// Mitsubishi GX Works2 project: 240909_공급가공   PLC: Q03UDV

PROGRAM MAIN
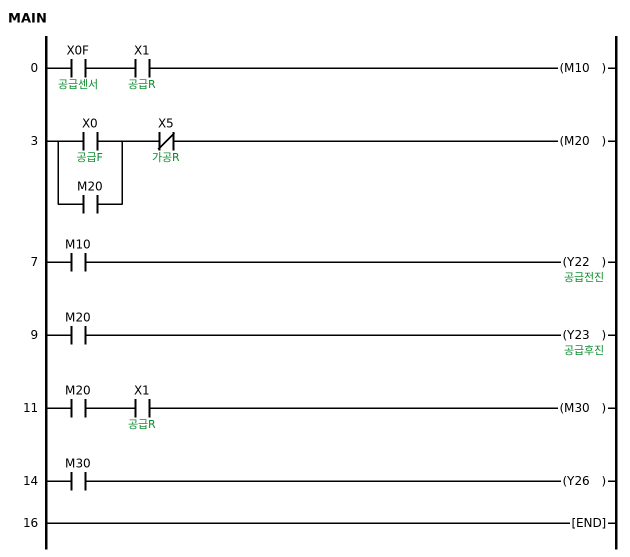
0     LD      X0F  ; 공급센서
      AND     X1  ; 공급R
      OUT     M10
3     LD      X0  ; 공급F
      OR      M20
      ANI     X5  ; 가공R
      OUT     M20
7     LD      M10
      OUT     Y22  ; 공급전진
9     LD      M20
      OUT     Y23  ; 공급후진
11    LD      M20
      AND     X1  ; 공급R
      OUT     M30
14    LD      M30
      OUT     Y26
16    END
END_PROGRAM
